// TIA Portal V20 export
FUNCTION_BLOCK "Kraft_Communication"   // FB3, LAD
{ S7_Optimized_Access := 'TRUE' }
// stored: MemoryReserve 100, SetENOAutomatically false
BEGIN
END_FUNCTION_BLOCK
